// TIA Portal V16 export
// export: Created 2024-12-03T15:41:42.7149112Z, ExportSetting WithDefaults, DisplayName Totally Integrated Automation Portal, DisplayVersion V16 Update 6, DisplayName TIA Portal Version Control Interface, DisplayVersion V16 Update 2, DisplayName TIA Portal Openness, DisplayVersion V16 Update 6, DisplayName TIA Portal Teamcenter Gateway, DisplayVersion V16, DisplayName SINAMICS Startdrive Advanced, DisplayVersion V16 Update 5, DisplayName SINAMICS Startdrive G130, G150, S120, S150, SINAMICS MV, S210, DisplayVersion V16 Update 5, DisplayName SINAMICS Startdrive G110M, G120, G120C, G120D, G120P, G115D, DisplayVersion V16 Update 5, DisplayName STEP 7 Professional, DisplayVersion V16 Update 6, DisplayName STEP 7 Safety, DisplayVersion V16, DisplayName WinCC Advanced / Unified PC, DisplayVersion V16 Update 6
FUNCTION_BLOCK "EvoLabel_FB"   // FB61, SCL
{ S7_Optimized_Access := 'TRUE' }
VERSION : 0.1
// stored: AutoNumber true, IsIECCheckEnabled false, IsRetainMemResEnabled false, MemoryReserve 100, SetENOAutomatically false, UDAEnableTagReadback false
   VAR_IN_OUT
      IO_EvoStatus : "EVO_LABEL_STATUS_UDT";
      IO_Printer : "EVO_LABEL_UDT";
   END_VAR
   VAR
      alarm : "AlarmInfo_UDT";
      offline { S7_SetPoint := 'True'} : "PLC_IPC_Status_FB";
      markerError { S7_SetPoint := 'True'} : "PLC_IPC_Status_FB";
      applicatorError { S7_SetPoint := 'True'} : "PLC_IPC_Status_FB";
      alarmOffline { S7_SetPoint := 'True'} : Program_Alarm;
      alarmMarker { S7_SetPoint := 'True'} : Program_Alarm;
      alarmApplicator { S7_SetPoint := 'True'} : Program_Alarm;
   END_VAR
   VAR_TEMP
      T_Appstate : "ApplicationState_UDT";
      T_Zone : "ZoneInfo";
   END_VAR
BEGIN
   REGION STATE
       #T_Zone := "ApplicationState_DB".ZoneNames[#IO_Printer.zone];
       #T_Appstate := "ApplicationState_DB".Appstate[#T_Zone.AppStateIndex];
   END_REGION

   REGION Build alarm info

       IF NOT #alarm.init OR #IO_Printer.name = '' OR #alarm.info = '' OR "HMI_DB".ReloadSettings.signal THEN

           #IO_Printer.name := "buildObjectName"(I_Symbolname := GetSymbolName(variable := #IO_Printer, size := 100));
           #alarm.info := "buildAlarmInfo"(I_ObjectName := #IO_Printer.name, I_ZoneIndex := #IO_Printer.zone, I_ZoneName := #T_Zone.ZoneName);
           #alarm.init := true;
       END_IF;

   END_REGION

   REGION ALARMS

       REGION PRINTER OFFLINE X0

           #offline(I_Reset := #T_Appstate.Hmi_Buttons.reset.state.LE,
                    O_Status => #IO_Printer.alarms.status.%X0,
                    IO_State := #IO_EvoStatus.online,
                    IO_Alarm := #IO_Printer.alarms.offline);

           #alarmOffline(SIG := #IO_Printer.alarms.offline,
                         SD_1 := #IO_Printer.name,
                         SD_2 := #T_Zone.ZoneName,
                         SD_3 := #alarm.info);

       END_REGION

       REGION PRINTER MARKER X1

           #markerError(I_Snooze := NOT #IO_EvoStatus.online,
                        I_Reset := #T_Appstate.Hmi_Buttons.reset.state.LE,
                        O_Status => #IO_Printer.alarms.status.%X1,
                        IO_State := #IO_EvoStatus.markerOk,
                        IO_Alarm := #IO_Printer.alarms.markerError);

           #alarmMarker(SIG := #IO_Printer.alarms.markerError,
                        SD_1 := #IO_Printer.name,
                        SD_2 := #T_Zone.ZoneName,
                        SD_3 := #alarm.info);

       END_REGION

       REGION PRINTER APPLICATOR X2

           #applicatorError(I_Snooze := NOT #IO_EvoStatus.online,
                            I_Reset := #T_Appstate.Hmi_Buttons.reset.state.LE,
                            O_Status => #IO_Printer.alarms.status.%X2,
                            IO_State := #IO_EvoStatus.applicatorOk,
                            IO_Alarm := #IO_Printer.alarms.applicatorError);

           #alarmApplicator(SIG := #IO_Printer.alarms.applicatorError,
                            SD_1 := #IO_Printer.name,
                            SD_2 := #T_Zone.ZoneName,
                            SD_3 := #alarm.info);

       END_REGION


       IF #IO_Printer.alarms.status > 0 THEN
           "ApplicationState_DB".Appstate[#T_Zone.AppStateIndex].Alarms.AlarmActiveInternalPLC := 1;
       END_IF;

   END_REGION
END_FUNCTION_BLOCK
